// TwinCAT 3 PLC project PLC
// ProgramVersion: 3.1.4024.0
// libraries:
//   Tc2_Standard, * (Beckhoff Automation GmbH)
//   Tc2_System, * (Beckhoff Automation GmbH)
//   Tc3_Module, * (Beckhoff Automation GmbH)
// project tree:
//   / PlcTask.TcTTO
//   POUs/ MAIN.TcPOU, Task1.TcPOU, Task2.TcPOU, Task3_GLV_HMI.TcPOU

CONFIGURATION PLC
    RESOURCE PLC ON TwinCAT3
        TASK PlcTask(INTERVAL := T#10ms, PRIORITY := 22);
        PROGRAM MAIN WITH PlcTask : MAIN;
    END_RESOURCE
END_CONFIGURATION

// ---- POUs/MAIN.TcPOU
PROGRAM MAIN
VAR
	fbArray:Task1;
	fbArrayCheck:Task2;
	fbPage:Task3_GLV_HMI;
END_VAR

fbArray();
fbArrayCheck();
fbPage();

END_PROGRAM

// ---- POUs/Task1.TcPOU
FUNCTION_BLOCK Task1
VAR_INPUT
END_VAR
VAR_OUTPUT
END_VAR
VAR
	aRandom : ARRAY[0..19] OF LREAL;  
	aMoved : ARRAY[0..19] OF LREAL; 
	aTest : ARRAY[0..19] OF LREAL; 
    i,j	: INT;                 
    lrRandValue: LREAL;
	Rand:DRAND;
	xGenerateOnce : BOOL := TRUE;
	iExecuteOnce : INT;
END_VAR

IF xGenerateOnce THEN
IF i=20 THEN // tu nie jesetem pewien, ale ten warunek jak zmienie na 19 to tablica generuje się w kółko, a przy 20 zmieniłem zakres tablicy na 20 i wartośc nie przypisała sie do tego 20 elementu,
		xGenerateOnce:=FALSE;
END_IF
	FOR i := 0 TO 19 BY 1 DO 
		Rand(Seed:= , Num=>lrRandValue );
    	aRandom[i] := lrRandValue*100;      
	END_FOR
END_IF

IF iExecuteOnce=0 THEN	
	MEMMOVE(destAddr := ADR(aMoved[1]), srcAddr := ADR(aRandom[0]), n := SIZEOF(aRandom) - SIZEOF(aRandom[0]));
	iExecuteOnce:=1;
END_IF

MEMMOVE(destAddr := ADR(aRandom), srcAddr := ADR(aMoved), n := SIZEOF(aMoved));
aRandom[0]:=1;

END_FUNCTION_BLOCK

// ---- POUs/Task2.TcPOU
FUNCTION_BLOCK Task2
VAR_INPUT
END_VAR
VAR_OUTPUT
END_VAR
VAR
	
	axTest : ARRAY[0..19] OF BOOL;
	i	:INT;
	
END_VAR

FOR i := 0 TO 19 BY 1 DO 	
	axTest[i]:= FALSE;
END_FOR
axTest[7]:= TRUE;

CheckIfAnyArrayElementIsTrue(axCheckTest:=axTest);

METHOD CheckIfAnyArrayElementIsTrue : BOOL
VAR_INPUT
	axCheckTest : ARRAY[0..19] OF BOOL;
END_VAR
VAR
	i	:INT;
	xCheck:BOOL;
END_VAR
VAR_INST
	xInArrayExistsTrueValue:BOOL;
END_VAR
FOR i := 0 TO 19 BY 1 DO 		
	
	IF axCheckTest[i] THEN
		
		xInArrayExistsTrueValue:=TRUE;
	
	ELSE
		;
	END_IF
	
END_FOR
END_METHOD

END_FUNCTION_BLOCK

// ---- POUs/Task3_GLV_HMI.TcPOU
FUNCTION_BLOCK Task3_GLV_HMI
VAR_INPUT
END_VAR
VAR_OUTPUT
END_VAR
VAR
	iPageNumber	:LREAL;

END_VAR

END_FUNCTION_BLOCK
